{attribute addProperty BoxType "EL5072-0000-0016"}
{attribute addProperty Id "UnderrangeBIT10.1251OverrangeBIT10.1252Excitation_errorBIT10.1253Input_errorBIT10.1254Digital_inputBIT10.1258Latch_extern_validBIT10.12510Set_position_doneBIT10.12511DiagBIT10.12513TxPDO_StateBIT10.12514Input_cycle_counter_BIT_0BIT10.12515Input_cycle_counter_BIT_1BIT10.12515"}
{attribute addProperty CRC "3775091545"}
{attribute addProperty SizeInBites "16"}
{attribute addProperty SizeInBytes "2"}
TYPE Status_E1035359 :
STRUCT
	{attribute addProperty Name "Underrange"}
	Underrange : BIT;
	{attribute addProperty Name "Overrange"}
	Overrange : BIT;
	{attribute addProperty Name "Excitation_error"}
	Excitation_error : BIT;
	{attribute addProperty Name "Input_error"}
	Input_error : BIT;
	{attribute 'hide'}
	reserve_1_BIT_0 : BIT;
	{attribute 'hide'}
	reserve_1_BIT_1 : BIT;
	{attribute 'hide'}
	reserve_1_BIT_2 : BIT;
	{attribute addProperty Name "Digital_input"}
	Digital_input : BIT;
	{attribute 'hide'}
	reserve_2 : BIT;
	{attribute addProperty Name "Latch_extern_valid"}
	Latch_extern_valid : BIT;
	{attribute addProperty Name "Set_position_done"}
	Set_position_done : BIT;
	{attribute 'hide'}
	reserve_3 : BIT;
	{attribute addProperty Name "Diag"}
	Diag : BIT;
	{attribute addProperty Name "TxPDO_State"}
	TxPDO_State : BIT;
	{attribute addProperty Name "Input_cycle_counter"}
	Input_cycle_counter_BIT_0 : BIT;
	{attribute addProperty Name "Input_cycle_counter"}
	Input_cycle_counter_BIT_1 : BIT;
END_STRUCT
END_TYPE

(* stored: Version 1.2.0.0, ProductVersion 3.1.4024.9
   DUT Status_E1035359: Id {f07a5ed0-bd6e-477b-bb65-5b39707dbf66} *)
